// TIA Portal project "2019" (V15.1)

(* hardware
DEVICE "S7300/ET200M station_1"  S7-300 station
   slot 0: "Rail_0"  Rail  6ES7 390-1***0-0AA0
   slot 2: "PLC_1"  CPU 314C-2 PN/DP  6ES7 314-6EH04-0AB0  V3.3
      slot 2: "PROFINET interface_1"  PN-IO
         slot 1: "Port_1"  Port
         slot 2: "Port_2"  Port
      slot 5: "DI 24/DO 16_1"  DI24/DO16
      slot 6: "AI 5/AO 2_1"  AI5/AO2
      slot 7: "Count_1"  Counter
      slot 8: "Positioning_1"  Positioning
   slot 4: "DO 8x24VDC/2A_1"  DO8 x 24VDC / 2A  6ES7 322-1BF01-0AA0
*)

// ===== PLC "PLC_1"  CPU 314C-2 PN/DP =====

VAR_GLOBAL   // PLC tag table "Default tag table"
   "F5" AT %I0.0 : Bool;
   "S3" AT %I0.1 : Bool;
   "S4" AT %I0.2 : Bool;
   "S5" AT %I0.3 : Bool;
   "S6" AT %I0.4 : Bool;
   "S7" AT %I0.5 : Bool;
   "S8" AT %I0.6 : Bool;
   "S9" AT %I0.7 : Bool;
   "S10" AT %I1.0 : Bool;
   "S11" AT %I1.1 : Bool;
   "Reserve1" AT %I1.2 : Bool;
   "BP1" AT %I1.3 : Bool;
   "B1" AT %I1.4 : Bool;
   "B2" AT %I1.5 : Bool;
   "Reserve2" AT %I1.6 : Bool;
   "B11" AT %I1.7 : Bool;
   "B12" AT %I2.0 : Bool;
   "B21" AT %I2.1 : Bool;
   "B22" AT %I2.2 : Bool;
   "B31" AT %I2.3 : Bool;
   "B32" AT %I2.4 : Bool;
   "Reserve3" AT %I2.5 : Bool;
   "Reserve4" AT %I2.6 : Bool;
   "Reserve5" AT %I2.7 : Bool;
   "M11" AT %Q0.0 : Bool;
   "M12" AT %Q0.1 : Bool;
   "M21" AT %Q0.2 : Bool;
   "M22" AT %Q0.3 : Bool;
   "M31" AT %Q0.4 : Bool;
   "M32" AT %Q0.5 : Bool;
   "Reserve6" AT %Q0.6 : Bool;
   "Reserve7" AT %Q0.7 : Bool;
   "P32" AT %Q1.0 : Bool;
   "P33" AT %Q1.1 : Bool;
   "Reserve8" AT %Q1.2 : Bool;
   "P2" AT %Q1.3 : Bool;
   "P3" AT %Q1.4 : Bool;
   "P4" AT %Q1.5 : Bool;
   "P5" AT %Q1.6 : Bool;
   "P6" AT %Q1.7 : Bool;
   "P7" AT %Q2.0 : Bool;
   "Reserve9" AT %Q2.1 : Bool;
   "P10" AT %Q2.2 : Bool;
   "P11" AT %Q2.3 : Bool;
   "P12" AT %Q2.4 : Bool;
   "P13" AT %Q2.5 : Bool;
   "P14" AT %Q2.6 : Bool;
   "P15" AT %Q2.7 : Bool;
   "active" AT %M0.0 : Bool;
END_VAR

DATA_BLOCK "Master_DB"   // DB1
{ S7_Optimized_Access := 'FALSE' }
VERSION : 0.1
// stored: InstanceOfName Master
"Master"
BEGIN
END_DATA_BLOCK

DATA_BLOCK "X2_DB"   // DB2
{ S7_Optimized_Access := 'FALSE' }
VERSION : 0.1
// stored: InstanceOfName Safety
"Safety"
BEGIN
END_DATA_BLOCK

DATA_BLOCK "G_Hienthi_DB"   // DB3
{ S7_Optimized_Access := 'FALSE' }
VERSION : 0.1
// stored: InstanceOfName G_Hienthi
"G_Hienthi"
BEGIN
END_DATA_BLOCK

DATA_BLOCK "1HZ_DB"   // DB6
{ S7_Optimized_Access := 'FALSE' }
VERSION : 0.1
// stored: InstanceOfName 1HZ
"1HZ"
BEGIN
END_DATA_BLOCK

DATA_BLOCK "G_Manual_DB"   // DB7
{ S7_Optimized_Access := 'FALSE' }
VERSION : 0.1
// stored: InstanceOfName G_Manual
"G_Manual"
BEGIN
END_DATA_BLOCK

DATA_BLOCK "G_Auto_DB"   // DB10
{ S7_Optimized_Access := 'FALSE' }
VERSION : 0.1
// stored: InstanceOfName G_Auto
"G_Auto"
BEGIN
END_DATA_BLOCK

DATA_BLOCK "output_DB"   // DB22
{ S7_Optimized_Access := 'FALSE' }
VERSION : 0.1
// stored: InstanceOfName output
"output"
BEGIN
END_DATA_BLOCK

FUNCTION_BLOCK "Master"   // FB1, FBD
{ S7_Optimized_Access := 'FALSE' }
VERSION : 0.1
   VAR_INPUT
      Activate : Bool;
      BP1 : Bool;
      S3 : Bool;
      S4 : Bool;
      F5 : Bool;
   END_VAR
   VAR_OUTPUT
      G_HIENTHI : Bool;
      Operation : Bool;
   END_VAR
   VAR
      X1 : Bool;
      X2 : Bool;
      X3 : Bool;
      X4 : Bool;
      X5 : Bool;
      P : Bool;
      MOperation : Bool;
   END_VAR
   VAR_TEMP   // added for the SCL form of the ladder/FBD networks
      _w1 : Bool;
   END_VAR
BEGIN

REGION Network 1
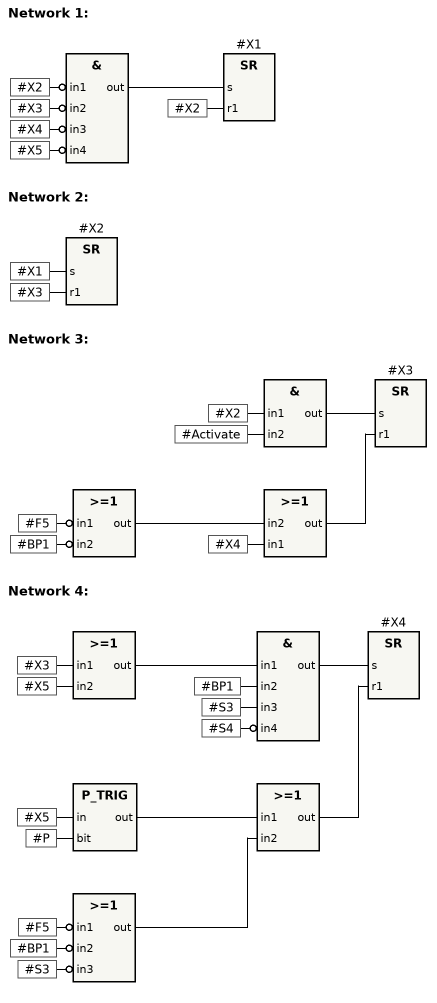
   IF NOT #X2 AND NOT #X3 AND NOT #X4 AND NOT #X5 THEN
       #X1 := TRUE;   // SR flip-flop
   END_IF;
   IF #X2 THEN #X1 := FALSE; END_IF;
END_REGION

REGION Network 2
   IF #X1 THEN
       #X2 := TRUE;   // SR flip-flop
   END_IF;
   IF #X3 THEN #X2 := FALSE; END_IF;
END_REGION

REGION Network 3
   IF #X2 AND #Activate THEN
       #X3 := TRUE;   // SR flip-flop
   END_IF;
   IF NOT #F5 OR NOT #BP1 OR #X4 THEN #X3 := FALSE; END_IF;
END_REGION

REGION Network 4
   #_w1 := #X5 AND NOT #P;   // rising edge
   #P := #X5;
   IF (#X3 OR #X5) AND #BP1 AND #S3 AND NOT #S4 THEN
       #X4 := TRUE;   // SR flip-flop
   END_IF;
   IF #_w1 OR NOT #F5 OR NOT #BP1 OR NOT #S3 THEN #X4 := FALSE; END_IF;
END_REGION

REGION Network 5
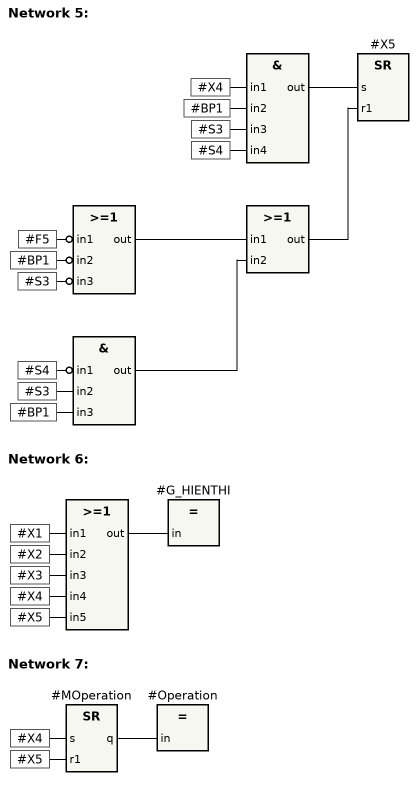
   IF #X4 AND #BP1 AND #S3 AND #S4 THEN
       #X5 := TRUE;   // SR flip-flop
   END_IF;
   IF NOT #F5 OR NOT #BP1 OR NOT #S3 OR (NOT #S4 AND #S3 AND #BP1) THEN #X5 := FALSE; END_IF;
END_REGION

REGION Network 6
   #G_HIENTHI := #X1 OR #X2 OR #X3 OR #X4 OR #X5;
END_REGION

REGION Network 7
   IF #X4 THEN
       #MOperation := TRUE;   // SR flip-flop
   END_IF;
   IF #X5 THEN #MOperation := FALSE; END_IF;
   #Operation := #MOperation;
END_REGION
END_FUNCTION_BLOCK

FUNCTION_BLOCK "Safety"   // FB2, FBD
{ S7_Optimized_Access := 'FALSE' }
VERSION : 0.1
   VAR_INPUT
      G_Kichhoat : Bool;
      F5 : Bool;
      S3 : Bool;
      S4 : Bool;
      S5 : Bool;
      S6 : Bool;
      S7 : Bool;
      S8 : Bool;
      S9 : Bool;
      S10 : Bool;
      S11 : Bool;
   END_VAR
   VAR_OUTPUT
      activate : Bool;
   END_VAR
   VAR
      X50 : Bool;
      X51 : Bool;
   END_VAR
BEGIN

REGION Network 1
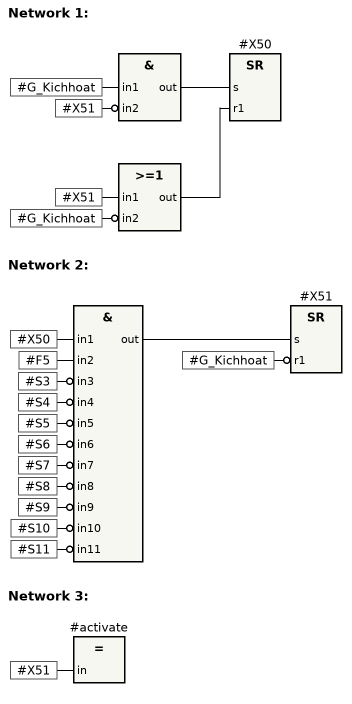
   IF #G_Kichhoat AND NOT #X51 THEN
       #X50 := TRUE;   // SR flip-flop
   END_IF;
   IF #X51 OR NOT #G_Kichhoat THEN #X50 := FALSE; END_IF;
END_REGION

REGION Network 2
   IF #X50 AND #F5 AND NOT #S3 AND NOT #S4 AND NOT #S5 AND NOT #S6 AND NOT #S7 AND NOT #S8 AND NOT #S9 AND NOT #S10 AND NOT #S11 THEN
       #X51 := TRUE;   // SR flip-flop
   END_IF;
   IF NOT #G_Kichhoat THEN #X51 := FALSE; END_IF;
END_REGION

REGION Network 3
   #activate := #X51;
END_REGION
END_FUNCTION_BLOCK

FUNCTION_BLOCK "G_Hienthi"   // FB3, FBD
{ S7_Optimized_Access := 'FALSE' }
VERSION : 0.1
   VAR_INPUT
      G_Hienthi : Bool;
      S3 : Bool;
      B12 : Bool;
      B22 : Bool;
      B32 : Bool;
      B1 : Bool;
      Operation : Bool;
      "Step" : Bool;
      BP1 : Bool;
      B11 : Bool;
      B21 : Bool;
      B31 : Bool;
      B2 : Bool;
   END_VAR
   VAR_OUTPUT
      P2 : Bool;
      P3 : Bool;
      P4 : Bool;
      P10 : Bool;
      P11 : Bool;
      P12 : Bool;
      P13 : Bool;
      P14 : Bool;
      P15 : Bool;
      P7 : Bool;
   END_VAR
   VAR
      X100 : Bool;
      X101 : Bool;
   END_VAR
BEGIN

REGION Network 1
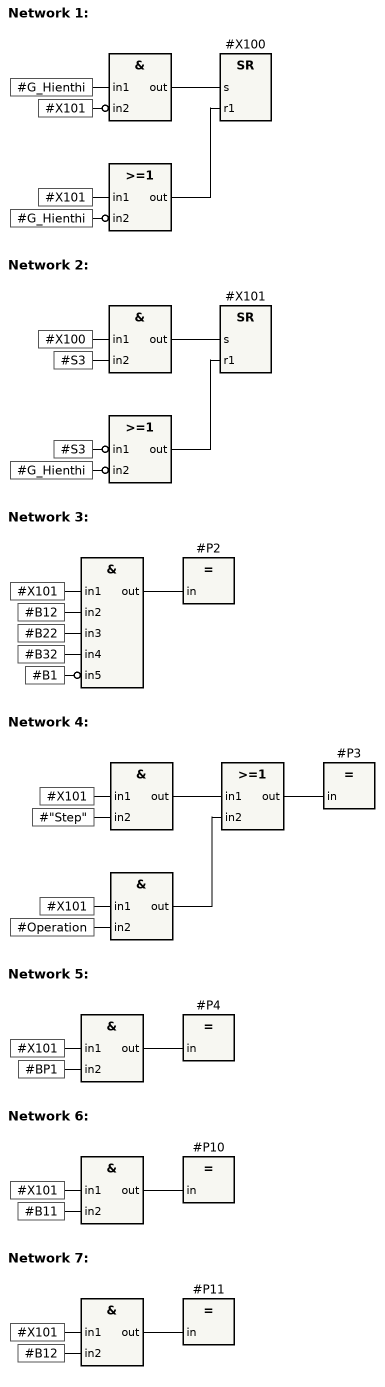
   IF #G_Hienthi AND NOT #X101 THEN
       #X100 := TRUE;   // SR flip-flop
   END_IF;
   IF #X101 OR NOT #G_Hienthi THEN #X100 := FALSE; END_IF;
END_REGION

REGION Network 2
   IF #X100 AND #S3 THEN
       #X101 := TRUE;   // SR flip-flop
   END_IF;
   IF NOT #S3 OR NOT #G_Hienthi THEN #X101 := FALSE; END_IF;
END_REGION

REGION Network 3
   #P2 := #X101 AND #B12 AND #B22 AND #B32 AND NOT #B1;
END_REGION

REGION Network 4
   #P3 := (#X101 AND #"Step") OR (#X101 AND #Operation);
END_REGION

REGION Network 5
   #P4 := #X101 AND #BP1;
END_REGION

REGION Network 6
   #P10 := #X101 AND #B11;
END_REGION

REGION Network 7
   #P11 := #X101 AND #B12;
END_REGION

REGION Network 8
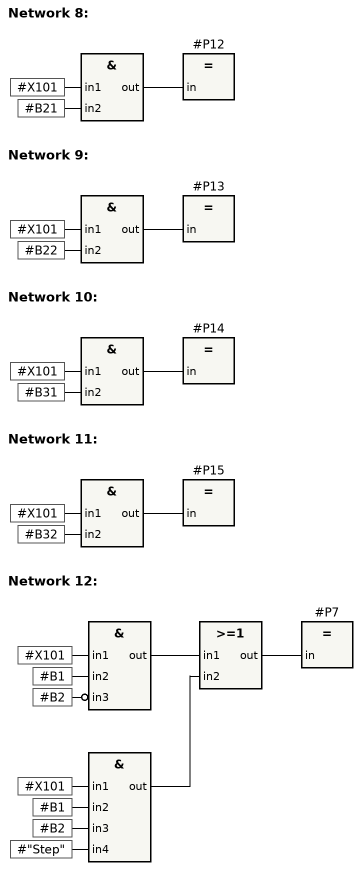
   #P12 := #X101 AND #B21;
END_REGION

REGION Network 9
   #P13 := #X101 AND #B22;
END_REGION

REGION Network 10
   #P14 := #X101 AND #B31;
END_REGION

REGION Network 11
   #P15 := #X101 AND #B32;
END_REGION

REGION Network 12
   #P7 := (#X101 AND #B1 AND NOT #B2) OR (#X101 AND #B1 AND #B2 AND #"Step");
END_REGION
END_FUNCTION_BLOCK

FUNCTION_BLOCK "1HZ"   // FB4, FBD
{ S7_Optimized_Access := 'FALSE' }
VERSION : 0.1
   VAR_OUTPUT
      "Step" : Bool;
   END_VAR
   VAR
      X200 : Bool;
      X201 : Bool;
      X202 : Bool;
   END_VAR
BEGIN

REGION Network 1
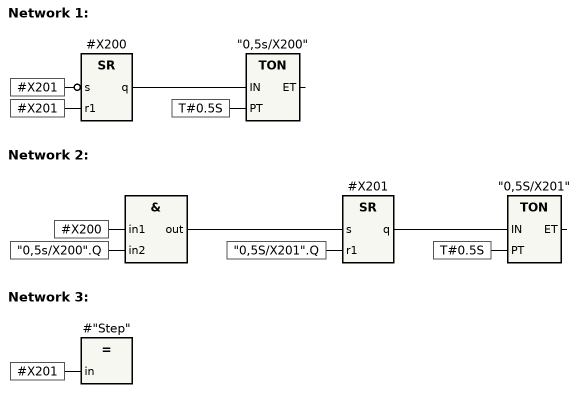
   IF NOT #X201 THEN
       #X200 := TRUE;   // SR flip-flop
   END_IF;
   IF #X201 THEN #X200 := FALSE; END_IF;
   "0,5s/X200".TON(IN := #X200, PT := T#0.5S);
END_REGION

REGION Network 2
   IF #X200 AND "0,5s/X200".Q THEN
       #X201 := TRUE;   // SR flip-flop
   END_IF;
   IF "0,5S/X201".Q THEN #X201 := FALSE; END_IF;
   "0,5S/X201".TON(IN := #X201, PT := T#0.5S);
END_REGION

REGION Network 3
   #"Step" := #X201;
END_REGION
END_FUNCTION_BLOCK

FUNCTION_BLOCK "G_Manual"   // FB5, FBD
{ S7_Optimized_Access := 'FALSE' }
VERSION : 0.1
   VAR_INPUT
      G_Manual : Bool;
      S6 : Bool;
      S7 : Bool;
      B11 : Bool;
      S8 : Bool;
      S9 : Bool;
      B21 : Bool;
      S10 : Bool;
      S11 : Bool;
      B31 : Bool;
      B12 : Bool;
      B22 : Bool;
      B32 : Bool;
   END_VAR
   VAR_OUTPUT
      M11 : Bool;
      M21 : Bool;
      M31 : Bool;
      M12 : Bool;
      M22 : Bool;
      M32 : Bool;
   END_VAR
   VAR
      X20 : Bool;
   END_VAR
BEGIN

REGION Network 1
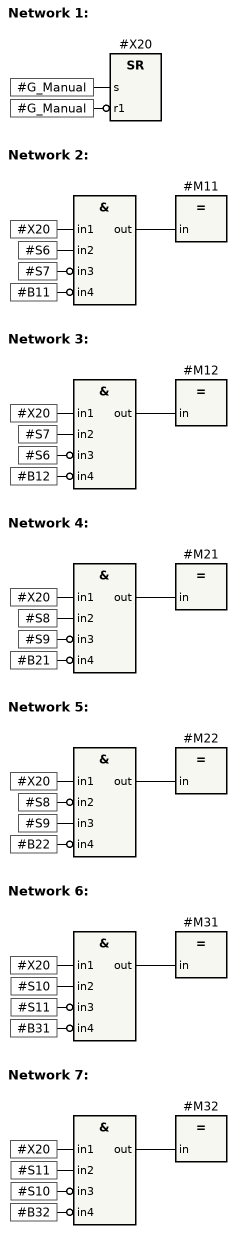
   IF #G_Manual THEN
       #X20 := TRUE;   // SR flip-flop
   END_IF;
   IF NOT #G_Manual THEN #X20 := FALSE; END_IF;
END_REGION

REGION Network 2
   #M11 := #X20 AND #S6 AND NOT #S7 AND NOT #B11;
END_REGION

REGION Network 3
   #M12 := #X20 AND #S7 AND NOT #S6 AND NOT #B12;
END_REGION

REGION Network 4
   #M21 := #X20 AND #S8 AND NOT #S9 AND NOT #B21;
END_REGION

REGION Network 5
   #M22 := #X20 AND NOT #S8 AND #S9 AND NOT #B22;
END_REGION

REGION Network 6
   #M31 := #X20 AND #S10 AND NOT #S11 AND NOT #B31;
END_REGION

REGION Network 7
   #M32 := #X20 AND #S11 AND NOT #S10 AND NOT #B32;
END_REGION
END_FUNCTION_BLOCK

FUNCTION_BLOCK "G_Auto"   // FB6, FBD
{ S7_Optimized_Access := 'FALSE' }
VERSION : 0.1
   VAR_INPUT
      G_Auto : Bool;
      "G_Safety.X50" : Bool;
      S5 : Bool;
      Operation : Bool;
      B11 : Bool;
      B12 : Bool;
      B1 : Bool;
      B2 : Bool;
      B31 : Bool;
      B21 : Bool;
      P2 : Bool;
   END_VAR
   VAR_OUTPUT
      P6 : Bool;
      P32 : Bool;
      P33 : Bool;
      M11 : Bool;
      M12 : Bool;
      M31 : Bool;
      M32 : Bool;
      M21 : Bool;
      M22 : Bool;
      P5 : Bool;
   END_VAR
   VAR
      X60 : Bool;
      X61 : Bool;
      X62 : Bool;
      X63 : Bool;
      X64 : Bool;
      X64A : Bool;
      X65 : Bool;
      X66 : Bool;
      X67 : Bool;
      X68 : Bool;
      X69 : Bool;
      "Phoi co" : Bool;
      Variable : Int;
      MWP : Bool;
      MP6 : Bool;
      MP32 : Bool;
      MP33 : Bool;
      P : Bool;
   END_VAR
   VAR_TEMP   // added for the SCL form of the ladder/FBD networks
      _w1 : Bool;
   END_VAR
BEGIN

REGION Network 1
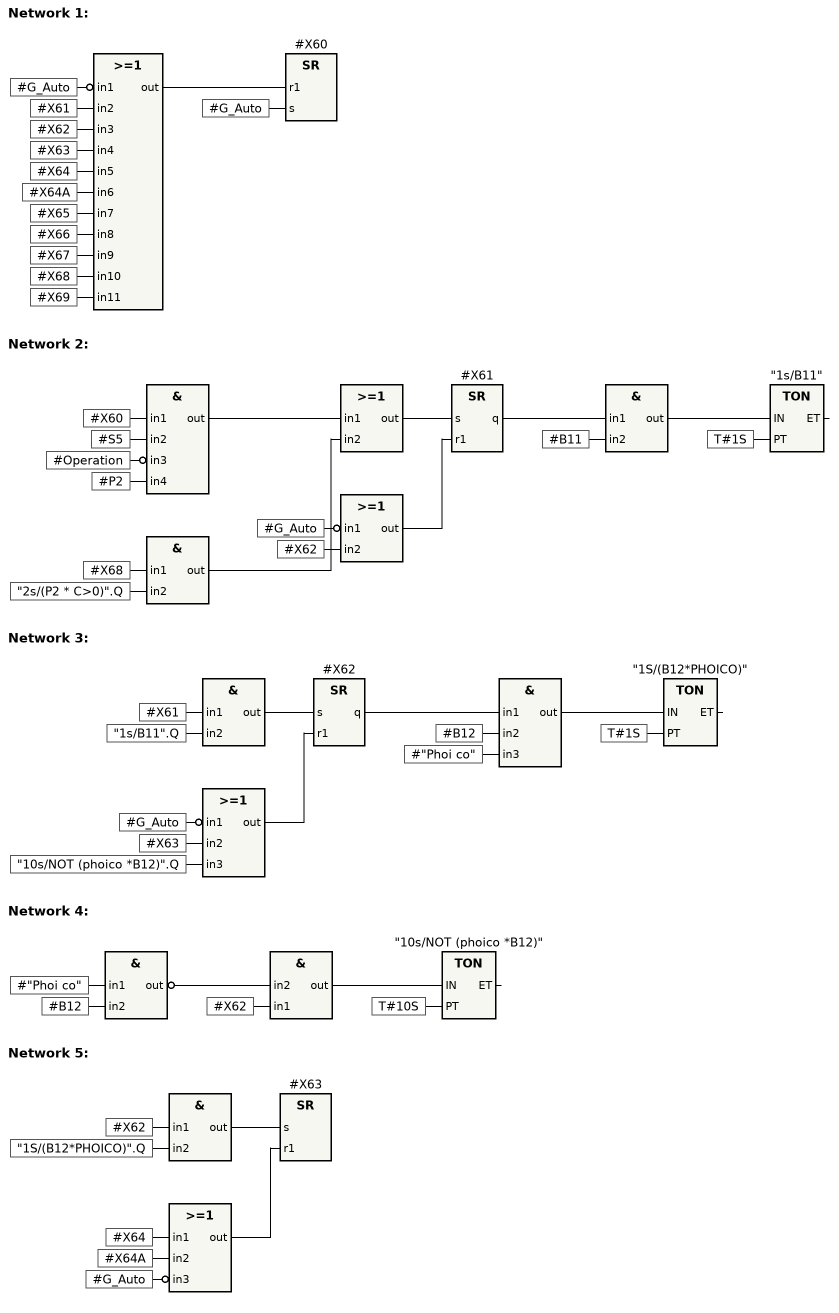
   IF #G_Auto THEN
       #X60 := TRUE;   // SR flip-flop
   END_IF;
   IF NOT #G_Auto OR #X61 OR #X62 OR #X63 OR #X64 OR #X64A OR #X65 OR #X66 OR #X67 OR #X68 OR #X69 THEN
       #X60 := FALSE;
   END_IF;
END_REGION

REGION Network 2
   IF (#X60 AND #S5 AND NOT #Operation AND #P2) OR (#X68 AND "2s/(P2 * C>0)".Q) THEN
       #X61 := TRUE;   // SR flip-flop
   END_IF;
   IF NOT #G_Auto OR #X62 THEN #X61 := FALSE; END_IF;
   "1s/B11".TON(IN := #X61 AND #B11, PT := T#1S);
END_REGION

REGION Network 3
   IF #X61 AND "1s/B11".Q THEN
       #X62 := TRUE;   // SR flip-flop
   END_IF;
   IF NOT #G_Auto OR #X63 OR "10s/NOT (phoico *B12)".Q THEN #X62 := FALSE; END_IF;
   "1S/(B12*PHOICO)".TON(IN := #X62 AND #B12 AND #"Phoi co", PT := T#1S);
END_REGION

REGION Network 4
   "10s/NOT (phoico *B12)".TON(IN := NOT (#"Phoi co" AND #B12) AND #X62, PT := T#10S);
END_REGION

REGION Network 5
   IF #X62 AND "1S/(B12*PHOICO)".Q THEN
       #X63 := TRUE;   // SR flip-flop
   END_IF;
   IF #X64 OR #X64A OR NOT #G_Auto THEN #X63 := FALSE; END_IF;
END_REGION

REGION Network 6
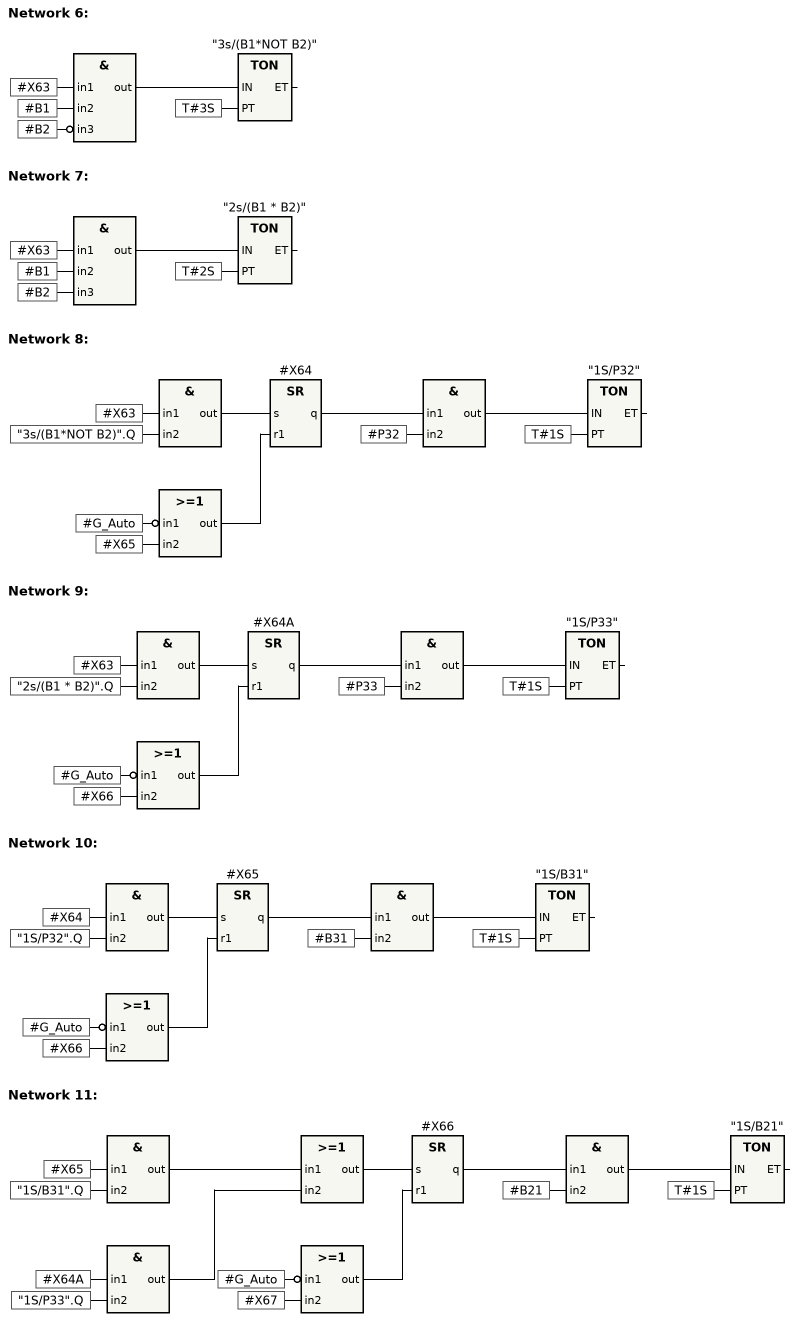
   "3s/(B1*NOT B2)".TON(IN := #X63 AND #B1 AND NOT #B2, PT := T#3S);
END_REGION

REGION Network 7
   "2s/(B1 * B2)".TON(IN := #X63 AND #B1 AND #B2, PT := T#2S);
END_REGION

REGION Network 8
   IF #X63 AND "3s/(B1*NOT B2)".Q THEN
       #X64 := TRUE;   // SR flip-flop
   END_IF;
   IF NOT #G_Auto OR #X65 THEN #X64 := FALSE; END_IF;
   "1S/P32".TON(IN := #X64 AND #P32, PT := T#1S);
END_REGION

REGION Network 9
   IF #X63 AND "2s/(B1 * B2)".Q THEN
       #X64A := TRUE;   // SR flip-flop
   END_IF;
   IF NOT #G_Auto OR #X66 THEN #X64A := FALSE; END_IF;
   "1S/P33".TON(IN := #X64A AND #P33, PT := T#1S);
END_REGION

REGION Network 10
   IF #X64 AND "1S/P32".Q THEN
       #X65 := TRUE;   // SR flip-flop
   END_IF;
   IF NOT #G_Auto OR #X66 THEN #X65 := FALSE; END_IF;
   "1S/B31".TON(IN := #X65 AND #B31, PT := T#1S);
END_REGION

REGION Network 11
   IF (#X65 AND "1S/B31".Q) OR (#X64A AND "1S/P33".Q) THEN
       #X66 := TRUE;   // SR flip-flop
   END_IF;
   IF NOT #G_Auto OR #X67 THEN #X66 := FALSE; END_IF;
   "1S/B21".TON(IN := #X66 AND #B21, PT := T#1S);
END_REGION

REGION Network 12
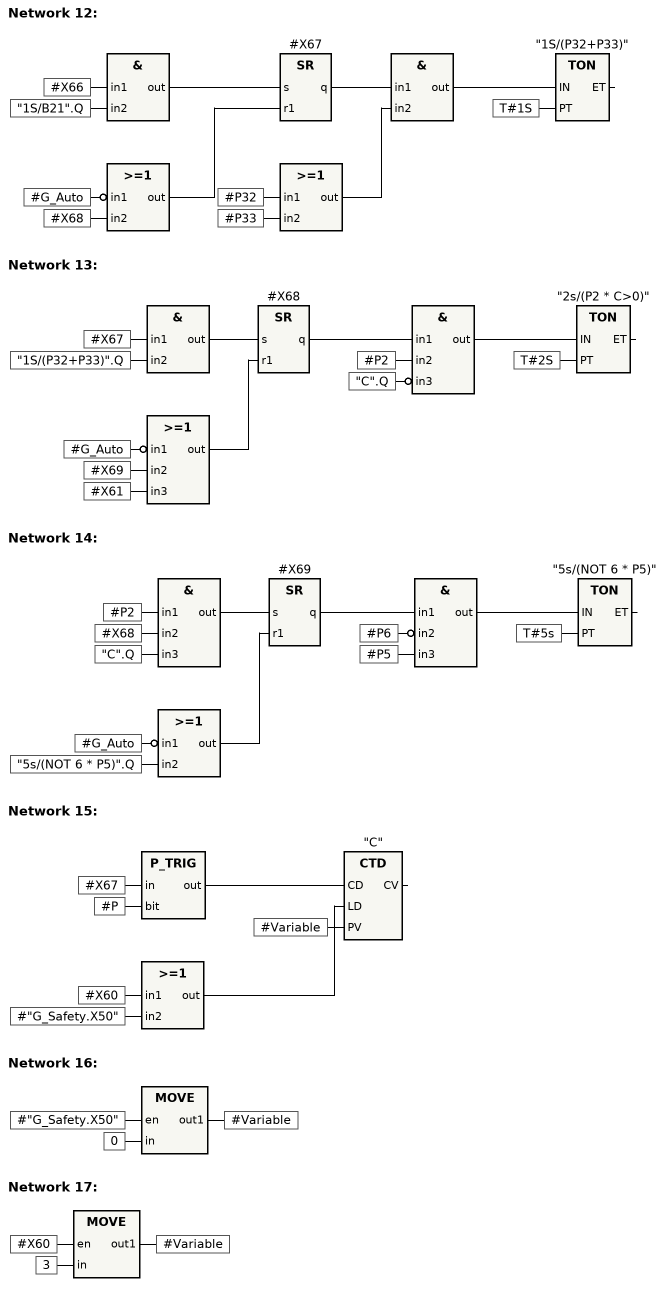
   IF #X66 AND "1S/B21".Q THEN
       #X67 := TRUE;   // SR flip-flop
   END_IF;
   IF NOT #G_Auto OR #X68 THEN #X67 := FALSE; END_IF;
   "1S/(P32+P33)".TON(IN := #X67 AND (#P32 OR #P33), PT := T#1S);
END_REGION

REGION Network 13
   IF #X67 AND "1S/(P32+P33)".Q THEN
       #X68 := TRUE;   // SR flip-flop
   END_IF;
   IF NOT #G_Auto OR #X69 OR #X61 THEN #X68 := FALSE; END_IF;
   "2s/(P2 * C>0)".TON(IN := #X68 AND #P2 AND NOT "C".Q, PT := T#2S);
END_REGION

REGION Network 14
   IF #P2 AND #X68 AND "C".Q THEN
       #X69 := TRUE;   // SR flip-flop
   END_IF;
   IF NOT #G_Auto OR "5s/(NOT 6 * P5)".Q THEN #X69 := FALSE; END_IF;
   "5s/(NOT 6 * P5)".TON(IN := #X69 AND NOT #P6 AND #P5, PT := T#5s);
END_REGION

REGION Network 15
   #_w1 := #X67 AND NOT #P;   // rising edge
   #P := #X67;
   "C".CTD(CD := #_w1, LD := #X60 OR #"G_Safety.X50", PV := #Variable);
END_REGION

REGION Network 16
   IF #"G_Safety.X50" THEN #Variable := 0; END_IF;
END_REGION

REGION Network 17
   IF #X60 THEN #Variable := 3; END_IF;
END_REGION

REGION Network 18
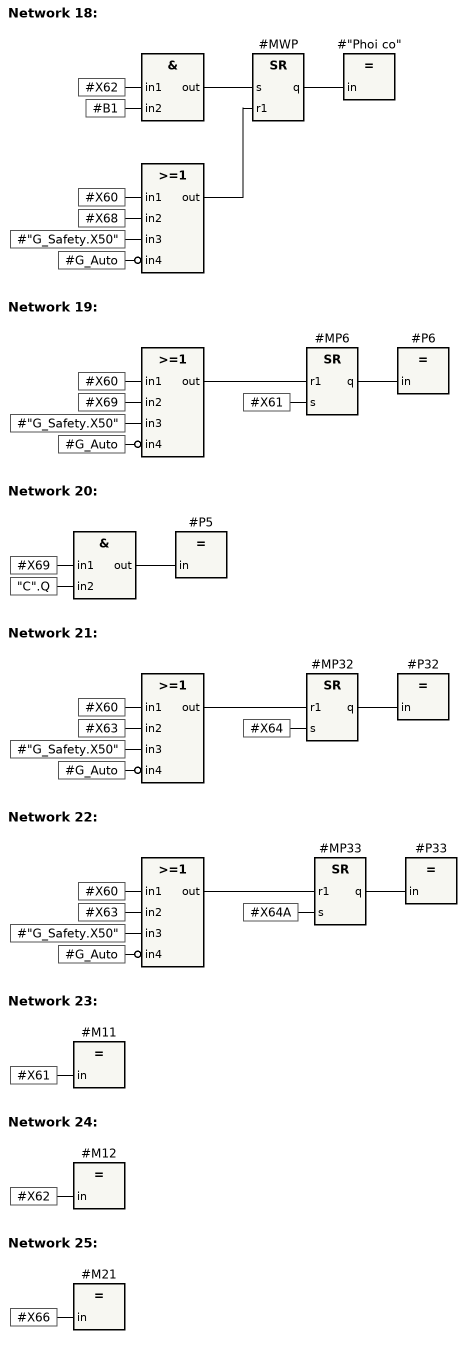
   IF #X62 AND #B1 THEN
       #MWP := TRUE;   // SR flip-flop
   END_IF;
   IF #X60 OR #X68 OR #"G_Safety.X50" OR NOT #G_Auto THEN #MWP := FALSE; END_IF;
   #"Phoi co" := #MWP;
END_REGION

REGION Network 19
   IF #X61 THEN
       #MP6 := TRUE;   // SR flip-flop
   END_IF;
   IF #X60 OR #X69 OR #"G_Safety.X50" OR NOT #G_Auto THEN #MP6 := FALSE; END_IF;
   #P6 := #MP6;
END_REGION

REGION Network 20
   #P5 := #X69 AND "C".Q;
END_REGION

REGION Network 21
   IF #X64 THEN
       #MP32 := TRUE;   // SR flip-flop
   END_IF;
   IF #X60 OR #X63 OR #"G_Safety.X50" OR NOT #G_Auto THEN #MP32 := FALSE; END_IF;
   #P32 := #MP32;
END_REGION

REGION Network 22
   IF #X64A THEN
       #MP33 := TRUE;   // SR flip-flop
   END_IF;
   IF #X60 OR #X63 OR #"G_Safety.X50" OR NOT #G_Auto THEN #MP33 := FALSE; END_IF;
   #P33 := #MP33;
END_REGION

REGION Network 23
   #M11 := #X61;
END_REGION

REGION Network 24
   #M12 := #X62;
END_REGION

REGION Network 25
   #M21 := #X66;
END_REGION

REGION Network 26
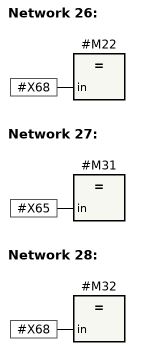
   #M22 := #X68;
END_REGION

REGION Network 27
   #M31 := #X65;
END_REGION

REGION Network 28
   #M32 := #X68;
END_REGION
END_FUNCTION_BLOCK

FUNCTION_BLOCK "output"   // FB7, FBD
{ S7_Optimized_Access := 'FALSE' }
VERSION : 0.1
   VAR_INPUT
      M11_A : Bool;
      M11_M : Bool;
      M12_A : Bool;
      M12_M : Bool;
      M21_A : Bool;
      M21_M : Bool;
      M22_A : Bool;
      M22_M : Bool;
      M31_A : Bool;
      M31_M : Bool;
      M32_A : Bool;
      M32_M : Bool;
   END_VAR
   VAR_OUTPUT
      M11 : Bool;
      M12 : Bool;
      M21 : Bool;
      M22 : Bool;
      M31 : Bool;
      M32 : Bool;
   END_VAR
BEGIN

REGION Network 1
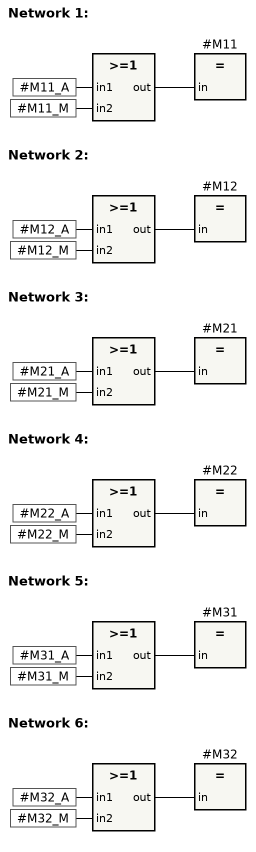
   #M11 := #M11_A OR #M11_M;
END_REGION

REGION Network 2
   #M12 := #M12_A OR #M12_M;
END_REGION

REGION Network 3
   #M21 := #M21_A OR #M21_M;
END_REGION

REGION Network 4
   #M22 := #M22_A OR #M22_M;
END_REGION

REGION Network 5
   #M31 := #M31_A OR #M31_M;
END_REGION

REGION Network 6
   #M32 := #M32_A OR #M32_M;
END_REGION
END_FUNCTION_BLOCK

ORGANIZATION_BLOCK "Main"   // OB1, FBD
TITLE = "Main Program Sweep (Cycle)"
{ S7_Optimized_Access := 'FALSE' }
VERSION : 0.1
   VAR_TEMP
      OB1_EV_CLASS : Byte;   // Bits 0-3 = 1 (Coming event), Bits 4-7 = 1 (Event class 1)
      OB1_SCAN_1 : Byte;   // 1 (Cold restart scan 1 of OB 1), 3 (Scan 2-n of OB 1)
      OB1_PRIORITY : Byte;   // Priority of OB Execution
      OB1_OB_NUMBR : Byte;   // 1 (Organization block 1, OB1)
      OB1_RESERVED_1 : Byte;   // Reserved for system
      OB1_RESERVED_2 : Byte;   // Reserved for system
      OB1_PREV_CYCLE : Int;   // Cycle time of previous OB1 scan (milliseconds)
      OB1_MIN_CYCLE : Int;   // Minimum cycle time of OB1 (milliseconds)
      OB1_MAX_CYCLE : Int;   // Maximum cycle time of OB1 (milliseconds)
      OB1_DATE_TIME : Date_And_Time;   // Date and time OB1 started
   END_VAR
BEGIN

REGION Network 1
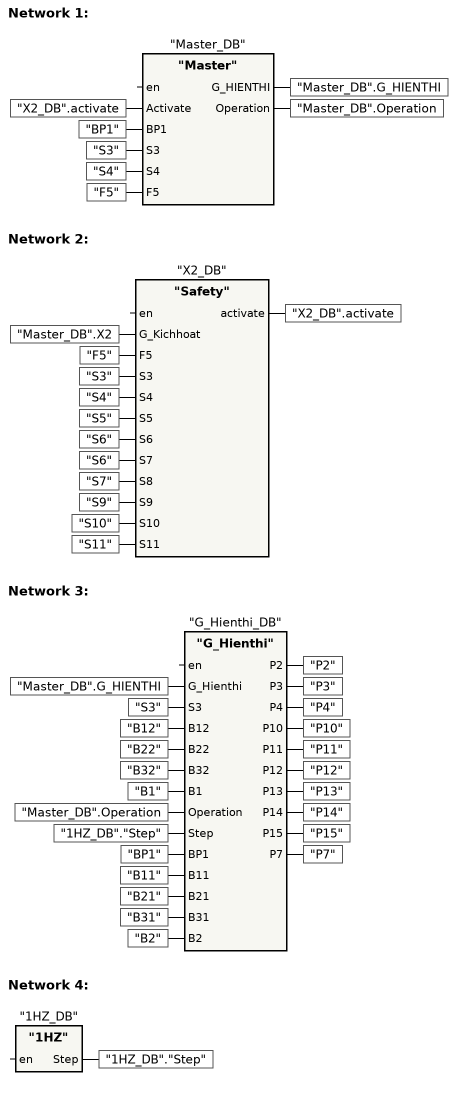
   "Master_DB"(Activate := "X2_DB".activate,   // "Master"
               BP1 := "BP1",
               S3 := "S3",
               S4 := "S4",
               F5 := "F5",
               G_HIENTHI => "Master_DB".G_HIENTHI,
               Operation => "Master_DB".Operation);
END_REGION

REGION Network 2
   "X2_DB"(G_Kichhoat := "Master_DB".X2,   // "Safety"
           F5 := "F5",
           S3 := "S3",
           S4 := "S4",
           S5 := "S5",
           S6 := "S6",
           S7 := "S6",
           S8 := "S7",
           S9 := "S9",
           S10 := "S10",
           S11 := "S11",
           activate => "X2_DB".activate);
END_REGION

REGION Network 3
   "G_Hienthi_DB"(G_Hienthi := "Master_DB".G_HIENTHI,   // "G_Hienthi"
                  S3 := "S3",
                  B12 := "B12",
                  B22 := "B22",
                  B32 := "B32",
                  B1 := "B1",
                  Operation := "Master_DB".Operation,
                  "Step" := "1HZ_DB"."Step",
                  BP1 := "BP1",
                  B11 := "B11",
                  B21 := "B21",
                  B31 := "B31",
                  B2 := "B2",
                  P2 => "P2",
                  P3 => "P3",
                  P4 => "P4",
                  P10 => "P10",
                  P11 => "P11",
                  P12 => "P12",
                  P13 => "P13",
                  P14 => "P14",
                  P15 => "P15",
                  P7 => "P7");
END_REGION

REGION Network 4
   "1HZ_DB"("Step" => "1HZ_DB"."Step");   // "1HZ"
END_REGION

REGION Network 5
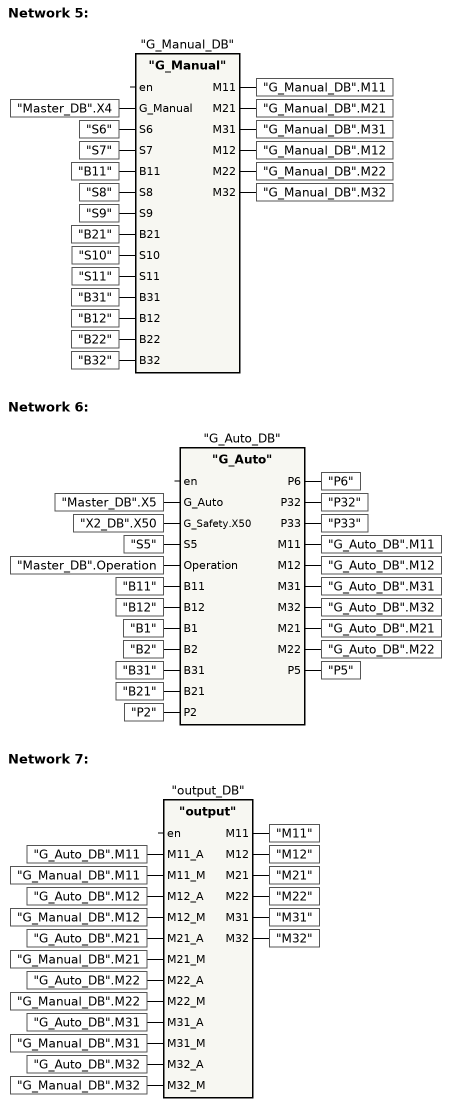
   "G_Manual_DB"(G_Manual := "Master_DB".X4,   // "G_Manual"
                 S6 := "S6",
                 S7 := "S7",
                 B11 := "B11",
                 S8 := "S8",
                 S9 := "S9",
                 B21 := "B21",
                 S10 := "S10",
                 S11 := "S11",
                 B31 := "B31",
                 B12 := "B12",
                 B22 := "B22",
                 B32 := "B32",
                 M11 => "G_Manual_DB".M11,
                 M21 => "G_Manual_DB".M21,
                 M31 => "G_Manual_DB".M31,
                 M12 => "G_Manual_DB".M12,
                 M22 => "G_Manual_DB".M22,
                 M32 => "G_Manual_DB".M32);
END_REGION

REGION Network 6
   "G_Auto_DB"(G_Auto := "Master_DB".X5,   // "G_Auto"
               "G_Safety.X50" := "X2_DB".X50,
               S5 := "S5",
               Operation := "Master_DB".Operation,
               B11 := "B11",
               B12 := "B12",
               B1 := "B1",
               B2 := "B2",
               B31 := "B31",
               B21 := "B21",
               P2 := "P2",
               P6 => "P6",
               P32 => "P32",
               P33 => "P33",
               M11 => "G_Auto_DB".M11,
               M12 => "G_Auto_DB".M12,
               M31 => "G_Auto_DB".M31,
               M32 => "G_Auto_DB".M32,
               M21 => "G_Auto_DB".M21,
               M22 => "G_Auto_DB".M22,
               P5 => "P5");
END_REGION

REGION Network 7
   "output_DB"(M11_A := "G_Auto_DB".M11,   // "output"
               M11_M := "G_Manual_DB".M11,
               M12_A := "G_Auto_DB".M12,
               M12_M := "G_Manual_DB".M12,
               M21_A := "G_Auto_DB".M21,
               M21_M := "G_Manual_DB".M21,
               M22_A := "G_Auto_DB".M22,
               M22_M := "G_Manual_DB".M22,
               M31_A := "G_Auto_DB".M31,
               M31_M := "G_Manual_DB".M31,
               M32_A := "G_Auto_DB".M32,
               M32_M := "G_Manual_DB".M32,
               M11 => "M11",
               M12 => "M12",
               M21 => "M21",
               M22 => "M22",
               M31 => "M31",
               M32 => "M32");
END_REGION
END_ORGANIZATION_BLOCK